{attribute 'linkalways'} 
{attribute 'no_explicit_call' := 'This FB is a CLASS and must be accessed using methods or properties'}
{attribute 'enable_dynamic_creation'}
FUNCTION_BLOCK FINAL SEL_LWORD EXTENDS Node
VAR
	g : _BOOL(FALSE);
	in1 : _LWORD(0);
	in2 : _LWORD(0);
	out : _LWORD(0);
END_VAR

METHOD PUBLIC Clone : I_Node
VAR
	pNode : POINTER TO SEL_LWORD;
END_VAR
pNode := __NEW(SEL_LWORD);
Clone := pNode^;
END_METHOD

METHOD FB_init : BOOL
VAR_INPUT
	bInitRetains : BOOL; // if TRUE, the retain variables are initialized (warm start / cold start)
	bInCopyCode : BOOL;  // if TRUE, the instance afterwards gets moved into the copy code (online change)
END_VAR
AddInput('g',THIS^.g);
AddInput('in1',THIS^.in1);
AddInput('in2',THIS^.in2);
AddOutput('out', THIS^.out);
END_METHOD

METHOD PROTECTED OnExecute
VAR
END_VAR
IF g.value THEN
	out.value := in2.value;
ELSE
	out.value := in1.value;
END_IF
END_METHOD

END_FUNCTION_BLOCK

(* stored: Version 1.1.0.1, ProductVersion 3.1.4024.15
   POU SEL_LWORD: Id {660ae2fa-9f67-4157-987d-80fc932dce68}, SpecialFunc None
   Folder Constructor: Id {99d606ff-0956-4a0e-8179-f8012d407af5}
   Method Clone: Id {897c3e98-8d30-45e7-af44-0b55757459fe}
   Method FB_init: Id {3cdf6522-ed47-47a7-8ed0-901c9f5c9dca}
   Method OnExecute: Id {79363c0e-d08f-4241-bf32-e8d1902c7915} *)
